PROGRAM MAIN
VAR
	// my comment
	a: BOOL := true;
	b: BOOL;
	c:bool;
END_VAR

a:=b;
c:=a;

END_PROGRAM

(* stored: Version 1.1.0.1, ProductVersion 3.1.0.25
   POU MAIN: Id {f4a86d2e-24eb-4ef3-a404-d704db804e38} *)
